# EPICS autosave request: utcaApp/Db/afc_timing_clock.req
$(P)$(R)$(CLOCK)FreqPropGain-SP
$(P)$(R)$(CLOCK)FreqIntgGain-SP
$(P)$(R)$(CLOCK)PhasePropGain-SP
$(P)$(R)$(CLOCK)PhaseIntgGain-SP
$(P)$(R)$(CLOCK)PhaseNavg-SP
$(P)$(R)$(CLOCK)PhaseDiv-SP
